(*
SPDX-FileCopyrightText: © 2026 Oleksandr Tiutyk <trofimich@gmail.com>
SPDX-License-Identifier: MIT
License: https://opensource.org/license/mit
*)

{attribute 'no_explicit_call' := 'do not call this function block directly'} 
PROGRAM GenericValueFactory
VAR_OUTPUT
	GenericValueClassName : STRING := 'GENERIC_VALUE';
END_VAR
VAR
	{attribute 'hide'} 
	_ClassName : STRING := __POUNAME();
END_VAR

{attribute 'monitoring' := 'call'}
PROPERTY ClassName : REFERENCE TO STRING
GET
ClassName REF= _ClassName;
END_GET
END_PROPERTY

METHOD FromAny : GENERIC_VALUE
VAR_INPUT
	value : ANY;
	isObject : BOOL;
	memoryManagementBehavior : GENERIC_MEMORY_MANAGEMENT_BEHAVIOR;
END_VAR
FromAny := FromAnyType(value, isObject, memoryManagementBehavior);
END_METHOD

METHOD FromAnyType : GENERIC_VALUE
VAR_INPUT
	value : __SYSTEM.AnyType;
	isObject : BOOL;
	memoryManagementBehavior : GENERIC_MEMORY_MANAGEMENT_BEHAVIOR;
END_VAR
FromAnyType := FromParts(GenericTypeClassConvertor.GetGenericTypeClassBySystemAnyType(value, isObject), value.pValue, TO_ULINT(value.diSize), memoryManagementBehavior);
END_METHOD

METHOD FromBoolReference : GENERIC_VALUE
VAR_IN_OUT
	value : BOOL;
END_VAR
FromBoolReference := FromParts(GENERIC_TYPE_CLASS.BOOLEAN, ADR(value), XSIZEOF(value), GENERIC_MEMORY_MANAGEMENT_BEHAVIOR.STORE_ORIGINAL_REFERENCE_AND_NOT_OWNS_MEMORY);
END_METHOD

METHOD FromBoolValue : GENERIC_VALUE
VAR_INPUT
	value : BOOL;
END_VAR
FromBoolValue := FromAny(value, FALSE, GENERIC_MEMORY_MANAGEMENT_BEHAVIOR.CLONE_ORIGINAL_VALUE_AND_OWNS_MEMORY);
END_METHOD

METHOD FromByteReference : GENERIC_VALUE
VAR_IN_OUT
	value : BYTE;
END_VAR
FromByteReference := FromParts(GENERIC_TYPE_CLASS.UINT_8, ADR(value), XSIZEOF(value), GENERIC_MEMORY_MANAGEMENT_BEHAVIOR.STORE_ORIGINAL_REFERENCE_AND_NOT_OWNS_MEMORY);
END_METHOD

METHOD FromByteValue : GENERIC_VALUE
VAR_INPUT
	value : BYTE;
END_VAR
FromByteValue := FromAny(value, FALSE, GENERIC_MEMORY_MANAGEMENT_BEHAVIOR.CLONE_ORIGINAL_VALUE_AND_OWNS_MEMORY);
END_METHOD

METHOD FromDateAndTimeReference : GENERIC_VALUE
VAR_IN_OUT
	value : DATE_AND_TIME;
END_VAR
FromDateAndTimeReference := FromParts(GENERIC_TYPE_CLASS.DATE_AND_TIME_32, ADR(value), XSIZEOF(value), GENERIC_MEMORY_MANAGEMENT_BEHAVIOR.STORE_ORIGINAL_REFERENCE_AND_NOT_OWNS_MEMORY);
END_METHOD

METHOD FromDateAndTimeValue : GENERIC_VALUE
VAR_INPUT
	value : DATE_AND_TIME;
END_VAR
FromDateAndTimeValue := FromAny(value, FALSE, GENERIC_MEMORY_MANAGEMENT_BEHAVIOR.CLONE_ORIGINAL_VALUE_AND_OWNS_MEMORY);
END_METHOD

METHOD FromDateReference : GENERIC_VALUE
VAR_IN_OUT
	value : DATE;
END_VAR
FromDateReference := FromParts(GENERIC_TYPE_CLASS.DATE_32, ADR(value), XSIZEOF(value), GENERIC_MEMORY_MANAGEMENT_BEHAVIOR.STORE_ORIGINAL_REFERENCE_AND_NOT_OWNS_MEMORY);
END_METHOD

METHOD FromDateValue : GENERIC_VALUE
VAR_INPUT
	value : DATE;
END_VAR
FromDateValue := FromAny(value, FALSE, GENERIC_MEMORY_MANAGEMENT_BEHAVIOR.CLONE_ORIGINAL_VALUE_AND_OWNS_MEMORY);
END_METHOD

METHOD FromDIntReference : GENERIC_VALUE
VAR_IN_OUT
	value : DINT;
END_VAR
FromDIntReference := FromParts(GENERIC_TYPE_CLASS.INT_32, ADR(value), XSIZEOF(value), GENERIC_MEMORY_MANAGEMENT_BEHAVIOR.STORE_ORIGINAL_REFERENCE_AND_NOT_OWNS_MEMORY);
END_METHOD

METHOD FromDIntValue : GENERIC_VALUE
VAR_INPUT
	value : DINT;
END_VAR
FromDIntValue := FromAny(value, FALSE, GENERIC_MEMORY_MANAGEMENT_BEHAVIOR.CLONE_ORIGINAL_VALUE_AND_OWNS_MEMORY);
END_METHOD

METHOD FromDWordReference : GENERIC_VALUE
VAR_IN_OUT
	value : DWORD;
END_VAR
FromDWordReference := FromParts(GENERIC_TYPE_CLASS.UINT_32, ADR(value), XSIZEOF(value), GENERIC_MEMORY_MANAGEMENT_BEHAVIOR.STORE_ORIGINAL_REFERENCE_AND_NOT_OWNS_MEMORY);
END_METHOD

METHOD FromDWordValue : GENERIC_VALUE
VAR_INPUT
	value : DWORD;
END_VAR
FromDWordValue := FromAny(value, FALSE, GENERIC_MEMORY_MANAGEMENT_BEHAVIOR.CLONE_ORIGINAL_VALUE_AND_OWNS_MEMORY);
END_METHOD

METHOD FromIntReference : GENERIC_VALUE
VAR_IN_OUT
	value : INT;
END_VAR
FromIntReference := FromParts(GENERIC_TYPE_CLASS.INT_16, ADR(value), XSIZEOF(value), GENERIC_MEMORY_MANAGEMENT_BEHAVIOR.STORE_ORIGINAL_REFERENCE_AND_NOT_OWNS_MEMORY);
END_METHOD

METHOD FromIntValue : GENERIC_VALUE
VAR_INPUT
	value : INT;
END_VAR
FromIntValue := FromAny(value, FALSE, GENERIC_MEMORY_MANAGEMENT_BEHAVIOR.CLONE_ORIGINAL_VALUE_AND_OWNS_MEMORY);
END_METHOD

METHOD FromIObjectReference : GENERIC_VALUE
VAR_INPUT
	instance : IObject;
END_VAR
VAR
	instanceNullException : ArgumentNotSpecifiedException;
END_VAR
IF instance = 0 THEN
	instanceNullException.Throw(NamespaceName, ClassName, __POUNAME(), __POSITION(), 'instance');
END_IF

FromIObjectReference := FromParts(GENERIC_TYPE_CLASS.OBJECT, instance.SelfAddress, instance.SelfSize, GENERIC_MEMORY_MANAGEMENT_BEHAVIOR.STORE_ORIGINAL_REFERENCE_AND_NOT_OWNS_MEMORY);
END_METHOD

METHOD FromIObjectValue : GENERIC_VALUE 
VAR_INPUT
	instance : IObject;
END_VAR
VAR
	instanceNullException : ArgumentNotSpecifiedException;

	cloneableIntance : ICloneable;
END_VAR
IF instance = 0 THEN
	instanceNullException.Throw(NamespaceName, ClassName, __POUNAME(), __POSITION(), 'instance');
END_IF

FromIObjectValue := FromParts(GENERIC_TYPE_CLASS.OBJECT, instance.SelfAddress, instance.SelfSize, GENERIC_MEMORY_MANAGEMENT_BEHAVIOR.CLONE_ORIGINAL_VALUE_AND_OWNS_MEMORY);
END_METHOD

METHOD FromLDateAndTimeReference : GENERIC_VALUE
VAR_IN_OUT
	value : LDATE_AND_TIME;
END_VAR
FromLDateAndTimeReference := FromParts(GENERIC_TYPE_CLASS.UINT_64, ADR(value), XSIZEOF(value), GENERIC_MEMORY_MANAGEMENT_BEHAVIOR.STORE_ORIGINAL_REFERENCE_AND_NOT_OWNS_MEMORY);
END_METHOD

METHOD FromLDateAndTimeValue : GENERIC_VALUE
VAR_INPUT
	value : LDATE_AND_TIME;
END_VAR
FromLDateAndTimeValue := FromAny(value, FALSE, GENERIC_MEMORY_MANAGEMENT_BEHAVIOR.CLONE_ORIGINAL_VALUE_AND_OWNS_MEMORY);
END_METHOD

METHOD FromLDateReference : GENERIC_VALUE
VAR_IN_OUT
	value : LDATE;
END_VAR
FromLDateReference := FromParts(GENERIC_TYPE_CLASS.UINT_64, ADR(value), XSIZEOF(value), GENERIC_MEMORY_MANAGEMENT_BEHAVIOR.STORE_ORIGINAL_REFERENCE_AND_NOT_OWNS_MEMORY);
END_METHOD

METHOD FromLDateValue : GENERIC_VALUE
VAR_INPUT
	value : LDATE;
END_VAR
FromLDateValue := FromAny(value, FALSE, GENERIC_MEMORY_MANAGEMENT_BEHAVIOR.CLONE_ORIGINAL_VALUE_AND_OWNS_MEMORY);
END_METHOD

METHOD FromLIntReference : GENERIC_VALUE
VAR_IN_OUT
	value : LINT;
END_VAR
FromLIntReference := FromParts(GENERIC_TYPE_CLASS.INT_64, ADR(value), XSIZEOF(value), GENERIC_MEMORY_MANAGEMENT_BEHAVIOR.STORE_ORIGINAL_REFERENCE_AND_NOT_OWNS_MEMORY);
END_METHOD

METHOD FromLIntValue : GENERIC_VALUE
VAR_INPUT
	value : LINT;
END_VAR
FromLIntValue := FromAny(value, FALSE, GENERIC_MEMORY_MANAGEMENT_BEHAVIOR.CLONE_ORIGINAL_VALUE_AND_OWNS_MEMORY);
END_METHOD

METHOD FromLRealReference : GENERIC_VALUE
VAR_IN_OUT
	value : LREAL;
END_VAR
FromLRealReference := FromParts(GENERIC_TYPE_CLASS.REAL_64, ADR(value), XSIZEOF(value), GENERIC_MEMORY_MANAGEMENT_BEHAVIOR.STORE_ORIGINAL_REFERENCE_AND_NOT_OWNS_MEMORY);
END_METHOD

METHOD FromLRealValue : GENERIC_VALUE
VAR_INPUT
	value : LREAL;
END_VAR
FromLRealValue := FromAny(value, FALSE, GENERIC_MEMORY_MANAGEMENT_BEHAVIOR.CLONE_ORIGINAL_VALUE_AND_OWNS_MEMORY);
END_METHOD

METHOD FromLTimeOfDayReference : GENERIC_VALUE
VAR_IN_OUT
	value : LTIME_OF_DAY;
END_VAR
FromLTimeOfDayReference := FromParts(GENERIC_TYPE_CLASS.UINT_64, ADR(value), XSIZEOF(value), GENERIC_MEMORY_MANAGEMENT_BEHAVIOR.STORE_ORIGINAL_REFERENCE_AND_NOT_OWNS_MEMORY);
END_METHOD

METHOD FromLTimeOfDayValue : GENERIC_VALUE
VAR_INPUT
	value : LTIME_OF_DAY;
END_VAR
FromLTimeOfDayValue := FromAny(value, FALSE, GENERIC_MEMORY_MANAGEMENT_BEHAVIOR.CLONE_ORIGINAL_VALUE_AND_OWNS_MEMORY);
END_METHOD

METHOD FromLTimeReference : GENERIC_VALUE
VAR_IN_OUT
	value : LTIME;
END_VAR
FromLTimeReference := FromParts(GENERIC_TYPE_CLASS.UINT_64, ADR(value), XSIZEOF(value), GENERIC_MEMORY_MANAGEMENT_BEHAVIOR.STORE_ORIGINAL_REFERENCE_AND_NOT_OWNS_MEMORY);
END_METHOD

METHOD FromLTimeValue : GENERIC_VALUE
VAR_INPUT
	value : LTIME;
END_VAR
FromLTimeValue := FromAny(value, FALSE, GENERIC_MEMORY_MANAGEMENT_BEHAVIOR.CLONE_ORIGINAL_VALUE_AND_OWNS_MEMORY);
END_METHOD

METHOD FromLWordReference : GENERIC_VALUE
VAR_IN_OUT
	value : LWORD;
END_VAR
FromLWordReference := FromParts(GENERIC_TYPE_CLASS.UINT_64, ADR(value), XSIZEOF(value), GENERIC_MEMORY_MANAGEMENT_BEHAVIOR.STORE_ORIGINAL_REFERENCE_AND_NOT_OWNS_MEMORY);
END_METHOD

METHOD FromLWordValue : GENERIC_VALUE
VAR_INPUT
	value : LWORD;
END_VAR
FromLWordValue := FromAny(value, FALSE, GENERIC_MEMORY_MANAGEMENT_BEHAVIOR.CLONE_ORIGINAL_VALUE_AND_OWNS_MEMORY);
END_METHOD

METHOD FromObjectReference : GENERIC_VALUE
VAR_INPUT
	instance : REFERENCE TO Object;
END_VAR
VAR
	instanceNullException : ArgumentNotSpecifiedException;
END_VAR
IF NOT __ISVALIDREF(instance) THEN
	instanceNullException.Throw(NamespaceName, ClassName, __POUNAME(), __POSITION(), 'instance');
END_IF

FromObjectReference := FromParts(GENERIC_TYPE_CLASS.OBJECT, instance.SelfAddress, instance.SelfSize, GENERIC_MEMORY_MANAGEMENT_BEHAVIOR.STORE_ORIGINAL_REFERENCE_AND_NOT_OWNS_MEMORY);
END_METHOD

METHOD FromObjectValue : GENERIC_VALUE 
VAR_INPUT
	instance : REFERENCE TO Object;
END_VAR
VAR
	instanceNullException : ArgumentNotSpecifiedException;

	cloneableIntance : ICloneable;
END_VAR
IF NOT __ISVALIDREF(instance) THEN
	instanceNullException.Throw(NamespaceName, ClassName, __POUNAME(), __POSITION(), 'instance');
END_IF

FromObjectValue := FromParts(GENERIC_TYPE_CLASS.OBJECT, instance.SelfAddress, instance.SelfSize, GENERIC_MEMORY_MANAGEMENT_BEHAVIOR.CLONE_ORIGINAL_VALUE_AND_OWNS_MEMORY);
END_METHOD

(*!
<summary>Creates a generic value from a type, address, size and memory-management policy.</summary>
<description>
Owning modes require permission to release the stored allocation, including any result returned by Clone.
Exception objects and their engine-managed clones are not supported by user-managed generic collections.
Their lifetime ends at cycle cleanup; use ERROR to retain an error as state.
</description>
*)
METHOD FromParts : GENERIC_VALUE
VAR_INPUT
	genericTypeClass : GENERIC_TYPE_CLASS;
	address : POINTER TO BYTE;
	size : ULINT;
	memoryManagementBehavior : GENERIC_MEMORY_MANAGEMENT_BEHAVIOR;
END_VAR
VAR
	newAddress : POINTER TO BYTE;

	objectPointer : POINTER TO Object;
	cloneable : ICloneable;
	clone : IObject;
END_VAR
IF address = 0 OR_ELSE size <= 0 THEN
	RETURN;
END_IF

CASE memoryManagementBehavior OF
	GENERIC_MEMORY_MANAGEMENT_BEHAVIOR.CLONE_ORIGINAL_VALUE_AND_OWNS_MEMORY:
		IF genericTypeClass = GENERIC_TYPE_CLASS.OBJECT THEN
			objectPointer := address;		
		END_IF
		
		IF genericTypeClass = GENERIC_TYPE_CLASS.OBJECT AND_THEN __QUERYINTERFACE(objectPointer^, cloneable) THEN
			clone := cloneable.Clone();
			newAddress := clone.SelfAddress;	
		ELSE
			newAddress := __NEW(BYTE, TO_UDINT(size));	
			Tc2_System.MEMCPY(newAddress, address, TO_UDINT(size));
		END_IF

		FromParts.Assign(genericTypeClass, newAddress, size, TRUE);
	
	GENERIC_MEMORY_MANAGEMENT_BEHAVIOR.STORE_ORIGINAL_REFERENCE_AND_NOT_OWNS_MEMORY:
		FromParts.Assign(genericTypeClass, address, size, FALSE);
	
	GENERIC_MEMORY_MANAGEMENT_BEHAVIOR.STORE_ORIGINAL_REFERENCE_AND_OWNS_MEMORY:
		FromParts.Assign(genericTypeClass, address, size, TRUE);
END_CASE
END_METHOD

METHOD FromRealReference : GENERIC_VALUE
VAR_IN_OUT
	value : REAL;
END_VAR
FromRealReference := FromParts(GENERIC_TYPE_CLASS.REAL_32, ADR(value), XSIZEOF(value), GENERIC_MEMORY_MANAGEMENT_BEHAVIOR.STORE_ORIGINAL_REFERENCE_AND_NOT_OWNS_MEMORY);
END_METHOD

METHOD FromRealValue : GENERIC_VALUE
VAR_INPUT
	value : REAL;
END_VAR
FromRealValue := FromAny(value, FALSE, GENERIC_MEMORY_MANAGEMENT_BEHAVIOR.CLONE_ORIGINAL_VALUE_AND_OWNS_MEMORY);
END_METHOD

METHOD FromSIntReference : GENERIC_VALUE
VAR_IN_OUT
	value : SINT;
END_VAR
FromSIntReference := FromParts(GENERIC_TYPE_CLASS.INT_8, ADR(value), XSIZEOF(value), GENERIC_MEMORY_MANAGEMENT_BEHAVIOR.STORE_ORIGINAL_REFERENCE_AND_NOT_OWNS_MEMORY);
END_METHOD

METHOD FromSIntValue : GENERIC_VALUE
VAR_INPUT
	value : SINT;
END_VAR
FromSIntValue := FromAny(value, FALSE, GENERIC_MEMORY_MANAGEMENT_BEHAVIOR.CLONE_ORIGINAL_VALUE_AND_OWNS_MEMORY);
END_METHOD

METHOD FromStringReference : GENERIC_VALUE
VAR_IN_OUT
	value : STRING;
END_VAR
FromStringReference := FromParts(GENERIC_TYPE_CLASS.STRING_ASCII, ADR(value), Strings.GetActualSize(value), GENERIC_MEMORY_MANAGEMENT_BEHAVIOR.STORE_ORIGINAL_REFERENCE_AND_NOT_OWNS_MEMORY);
END_METHOD

METHOD FromStringValue : GENERIC_VALUE
VAR_IN_OUT CONSTANT
	value : STRING;
END_VAR
FromStringValue := FromParts(GENERIC_TYPE_CLASS.STRING_ASCII, ADR(value), Strings.GetActualSize(value), GENERIC_MEMORY_MANAGEMENT_BEHAVIOR.CLONE_ORIGINAL_VALUE_AND_OWNS_MEMORY);
END_METHOD

METHOD FromTimeOfDayReference : GENERIC_VALUE
VAR_IN_OUT
	value : TIME_OF_DAY;
END_VAR
FromTimeOfDayReference := FromParts(GENERIC_TYPE_CLASS.TIME_OF_DAY_32, ADR(value), XSIZEOF(value), GENERIC_MEMORY_MANAGEMENT_BEHAVIOR.STORE_ORIGINAL_REFERENCE_AND_NOT_OWNS_MEMORY);
END_METHOD

METHOD FromTimeOfDayValue : GENERIC_VALUE
VAR_INPUT
	value : TIME_OF_DAY;
END_VAR
FromTimeOfDayValue := FromAny(value, FALSE, GENERIC_MEMORY_MANAGEMENT_BEHAVIOR.CLONE_ORIGINAL_VALUE_AND_OWNS_MEMORY);
END_METHOD

METHOD FromTimeReference : GENERIC_VALUE
VAR_IN_OUT
	value : TIME;
END_VAR
FromTimeReference := FromParts(GENERIC_TYPE_CLASS.TIME_32, ADR(value), XSIZEOF(value), GENERIC_MEMORY_MANAGEMENT_BEHAVIOR.STORE_ORIGINAL_REFERENCE_AND_NOT_OWNS_MEMORY);
END_METHOD

METHOD FromTimeValue : GENERIC_VALUE
VAR_INPUT
	value : TIME;
END_VAR
FromTimeValue := FromAny(value, FALSE, GENERIC_MEMORY_MANAGEMENT_BEHAVIOR.CLONE_ORIGINAL_VALUE_AND_OWNS_MEMORY);
END_METHOD

METHOD FromUDIntReference : GENERIC_VALUE
VAR_IN_OUT
	value : UDINT;
END_VAR
FromUDIntReference := FromParts(GENERIC_TYPE_CLASS.UINT_32, ADR(value), XSIZEOF(value), GENERIC_MEMORY_MANAGEMENT_BEHAVIOR.STORE_ORIGINAL_REFERENCE_AND_NOT_OWNS_MEMORY);
END_METHOD

METHOD FromUDIntValue : GENERIC_VALUE
VAR_INPUT
	value : UDINT;
END_VAR
FromUDIntValue := FromAny(value, FALSE, GENERIC_MEMORY_MANAGEMENT_BEHAVIOR.CLONE_ORIGINAL_VALUE_AND_OWNS_MEMORY);
END_METHOD

METHOD FromUIntReference : GENERIC_VALUE
VAR_IN_OUT
	value : UINT;
END_VAR
FromUIntReference := FromParts(GENERIC_TYPE_CLASS.UINT_16, ADR(value), XSIZEOF(value), GENERIC_MEMORY_MANAGEMENT_BEHAVIOR.STORE_ORIGINAL_REFERENCE_AND_NOT_OWNS_MEMORY);
END_METHOD

METHOD FromUIntValue : GENERIC_VALUE
VAR_INPUT
	value : UINT;
END_VAR
FromUIntValue := FromAny(value, FALSE, GENERIC_MEMORY_MANAGEMENT_BEHAVIOR.CLONE_ORIGINAL_VALUE_AND_OWNS_MEMORY);
END_METHOD

METHOD FromULIntReference : GENERIC_VALUE
VAR_IN_OUT
	value : ULINT;
END_VAR
FromULIntReference := FromParts(GENERIC_TYPE_CLASS.UINT_64, ADR(value), XSIZEOF(value), GENERIC_MEMORY_MANAGEMENT_BEHAVIOR.STORE_ORIGINAL_REFERENCE_AND_NOT_OWNS_MEMORY);
END_METHOD

METHOD FromULIntValue : GENERIC_VALUE
VAR_INPUT
	value : ULINT;
END_VAR
FromULIntValue := FromAny(value, FALSE, GENERIC_MEMORY_MANAGEMENT_BEHAVIOR.CLONE_ORIGINAL_VALUE_AND_OWNS_MEMORY);
END_METHOD

METHOD FromUSIntReference : GENERIC_VALUE
VAR_IN_OUT
	value : USINT;
END_VAR
FromUSIntReference := FromParts(GENERIC_TYPE_CLASS.UINT_8, ADR(value), XSIZEOF(value), GENERIC_MEMORY_MANAGEMENT_BEHAVIOR.STORE_ORIGINAL_REFERENCE_AND_NOT_OWNS_MEMORY);
END_METHOD

METHOD FromUSIntValue : GENERIC_VALUE
VAR_INPUT
	value : USINT;
END_VAR
FromUSIntValue := FromAny(value, FALSE, GENERIC_MEMORY_MANAGEMENT_BEHAVIOR.CLONE_ORIGINAL_VALUE_AND_OWNS_MEMORY);
END_METHOD

METHOD FromWordReference : GENERIC_VALUE
VAR_IN_OUT
	value : WORD;
END_VAR
FromWordReference := FromParts(GENERIC_TYPE_CLASS.UINT_16, ADR(value), XSIZEOF(value), GENERIC_MEMORY_MANAGEMENT_BEHAVIOR.STORE_ORIGINAL_REFERENCE_AND_NOT_OWNS_MEMORY);
END_METHOD

METHOD FromWordValue : GENERIC_VALUE
VAR_INPUT
	value : WORD;
END_VAR
FromWordValue := FromAny(value, FALSE, GENERIC_MEMORY_MANAGEMENT_BEHAVIOR.CLONE_ORIGINAL_VALUE_AND_OWNS_MEMORY);
END_METHOD

METHOD FromWStringReference : GENERIC_VALUE
VAR_IN_OUT
	value : WSTRING;
END_VAR
FromWStringReference := FromParts(GENERIC_TYPE_CLASS.STRING_UTF16, ADR(value), WideStrings.GetActualSize(value), GENERIC_MEMORY_MANAGEMENT_BEHAVIOR.STORE_ORIGINAL_REFERENCE_AND_NOT_OWNS_MEMORY);
END_METHOD

METHOD FromWStringValue : GENERIC_VALUE
VAR_IN_OUT CONSTANT
	value : WSTRING;
END_VAR
FromWStringValue := FromParts(GENERIC_TYPE_CLASS.STRING_UTF16, ADR(value), WideStrings.GetActualSize(value), GENERIC_MEMORY_MANAGEMENT_BEHAVIOR.CLONE_ORIGINAL_VALUE_AND_OWNS_MEMORY);
END_METHOD

{attribute 'monitoring' := 'call'}
PROPERTY NamespaceName : REFERENCE TO STRING
GET
NamespaceName REF= CurrentNamespace.Name;
END_GET
END_PROPERTY

END_PROGRAM

(* stored: Version 1.1.0.1
   POU GenericValueFactory: Id {5aafca66-5cdb-4882-83ad-05bcd6342c33}, SpecialFunc None
   Folder FromTypedReferences: Id {6a62176f-75b8-40f9-88f4-26d2c66b2b4c}
   Folder Date and time: Id {50be7849-3dc1-473b-9a05-6b6e31d6af8b}
   Folder Floating point: Id {135cf303-d7c8-4cb2-83e4-8818dc564814}
   Folder Integer: Id {9822276d-d405-467b-913a-d88d688e27ab}
   Folder Signed: Id {88769d57-d90b-4d86-a952-5ee7177698c2}
   Folder Unsugned: Id {b4e483f8-ba35-4ef4-8231-cc40ee080b19}
   Folder Strings: Id {eee688c5-eebb-4825-a4d2-c0399523c8d1}
   Folder FromTypedValues: Id {25ae72e5-a435-4f95-b7ff-4fa29bd648e4}
   Folder Date and time: Id {c40440d3-8031-4729-9442-ab1c6e1a88ce}
   Folder Floating point: Id {87a9bf3e-1364-4eb7-acac-0cdf6af21cc8}
   Folder Integer: Id {0a1aa935-644b-4556-94c3-416eb3400fa0}
   Folder Signed: Id {940b3a7d-41f9-44cf-8d1e-ff10f12d8a45}
   Folder Unsugned: Id {0879f3ef-e520-4036-bc27-14c1b4a89e4e}
   Folder Strings: Id {b9fa53fd-8c54-4f18-b477-b593285e3922}
   Property ClassName: Id {471a3424-a03f-46e9-aa5d-47ddfd6d5482}
   Get Get: Id {a20ec758-d80c-4890-b9c6-9d76856ede75}
   Method FromAny: Id {6ea8f682-f65a-4f72-b981-df5fc5f1ef43}
   Method FromAnyType: Id {58f5fed2-ee58-4bb7-b5fb-7380db0fc95f}
   Method FromBoolReference: Id {d27b6912-bb8f-448c-b703-74f93763bb2a}
   Method FromBoolValue: Id {05323a56-8230-4256-ab0d-6fb067ae3a7c}
   Method FromByteReference: Id {d0163973-28dc-453e-ad54-13cb227a8692}
   Method FromByteValue: Id {c850b1be-a21b-48c4-b41a-36d350dde20f}
   Method FromDateAndTimeReference: Id {173ac213-1cc9-43cb-af55-055a2d088a5d}
   Method FromDateAndTimeValue: Id {acb7264d-a9f1-46b1-a8df-1b273f60647d}
   Method FromDateReference: Id {e4aa20a7-899e-4891-8b7b-4b75565ece84}
   Method FromDateValue: Id {23c94b95-80f9-479f-a2c5-e7d679fc27d6}
   Method FromDIntReference: Id {347f607f-2c78-4202-8506-027cbef4c70e}
   Method FromDIntValue: Id {3180b989-96c3-434b-b481-bd0a4f94dfea}
   Method FromDWordReference: Id {946efa8e-2ab5-43b1-bf77-3303cffc04cb}
   Method FromDWordValue: Id {a4f9425d-c238-4587-bc3b-6ca752d58eb9}
   Method FromIntReference: Id {297f6b14-cf53-4dfc-8218-a8424a5edfe0}
   Method FromIntValue: Id {8dbf331d-d65d-4447-810a-b5722dd5340b}
   Method FromIObjectReference: Id {5e9ad193-b039-42bb-8395-af4a1c647cfc}
   Method FromIObjectValue: Id {fef270e2-21e0-469c-8151-9d5a311dfd4b}
   Method FromLDateAndTimeReference: Id {73c19958-a0a7-4e2d-ade2-e984449c3d1d}
   Method FromLDateAndTimeValue: Id {a766e905-b94b-4c9d-82d2-dc889e57d0b8}
   Method FromLDateReference: Id {580e428d-fb4b-4375-874d-309e30a280bf}
   Method FromLDateValue: Id {3521f0fd-d786-4c9e-9852-33d078c765f7}
   Method FromLIntReference: Id {3587c5a4-e047-430d-a163-142a19047459}
   Method FromLIntValue: Id {60a27329-0eea-455a-849b-eb1a0f8b3d54}
   Method FromLRealReference: Id {b3eac24c-b062-484b-ad9a-bc37b94b04ce}
   Method FromLRealValue: Id {3dd0d52e-c433-4065-9057-391e0b5d7161}
   Method FromLTimeOfDayReference: Id {ddcd78a1-0fee-4add-a56e-178a6a711394}
   Method FromLTimeOfDayValue: Id {383c7178-c7ae-4a60-9f1e-7d0d454ddfe1}
   Method FromLTimeReference: Id {09bff33e-4edf-4b18-8976-6a561c6f9e70}
   Method FromLTimeValue: Id {720ca242-94c2-488a-8631-0658baa256f2}
   Method FromLWordReference: Id {f772b6da-0878-4a66-aae9-b922e2dd49f9}
   Method FromLWordValue: Id {1b4080c1-48c3-4e24-89fd-b9ed03b1ebe8}
   Method FromObjectReference: Id {1f38a672-fb8f-436c-9ddd-df1d9f011e0c}
   Method FromObjectValue: Id {ad024805-1158-4b96-998d-e6f1c85f0eb0}
   Method FromParts: Id {759e0037-660d-404f-8404-ca0ffa255f71}
   Method FromRealReference: Id {3b55838d-58fe-4935-bf92-dcc94945943e}
   Method FromRealValue: Id {f5d5afa5-da33-48d8-929b-a1880a20b6ed}
   Method FromSIntReference: Id {dcbeabb7-7a7d-43d2-8ece-e53719a456af}
   Method FromSIntValue: Id {69dc6169-e00d-4a1b-a310-c30817210f3f}
   Method FromStringReference: Id {ab2c82b3-b73e-4926-9fa1-21180356ffa0}
   Method FromStringValue: Id {a2ca4991-d75a-4278-817b-66b69acc26fd}
   Method FromTimeOfDayReference: Id {16667815-ae24-4a2e-bb7e-13b02852bf9b}
   Method FromTimeOfDayValue: Id {e882c6af-473d-4d99-a60c-86a44c55080d}
   Method FromTimeReference: Id {4efbab6a-08c6-45a2-8741-5970c5b4615c}
   Method FromTimeValue: Id {9ee9b713-8171-4acb-a940-5ccce35b7698}
   Method FromUDIntReference: Id {1c502058-ad42-4bc4-99e4-7e76741e1405}
   Method FromUDIntValue: Id {168c3430-037e-43ee-96ec-29f9d4ddb82b}
   Method FromUIntReference: Id {81d69bd9-3d0f-4fa9-a701-f3d6b82d40a5}
   Method FromUIntValue: Id {92156321-3e30-463a-83fa-c306bca1bc5c}
   Method FromULIntReference: Id {a686507f-51c4-410e-98ad-c2541ef602d2}
   Method FromULIntValue: Id {86c92bb6-733a-407c-aa95-3d976887e765}
   Method FromUSIntReference: Id {946118fe-852d-4783-9124-b28f9c5aa505}
   Method FromUSIntValue: Id {aeae6bc1-69d5-4f8e-bf8c-5456e7fca1c3}
   Method FromWordReference: Id {3a044499-0651-4e47-8802-27ec81f73705}
   Method FromWordValue: Id {cf646851-d26b-43e6-9a97-f0629adff38e}
   Method FromWStringReference: Id {ef6f17c2-c854-4bd1-98d9-b20dcef69d2f}
   Method FromWStringValue: Id {7495b560-9d45-42dd-b7ac-cea5caf03cd8}
   Property NamespaceName: Id {1b7a4363-1ae3-4082-9387-38baaafa2b6f}
   Get Get: Id {d9491450-ccd1-4cff-a47e-d13d4898b8f0} *)
